// TIA Portal V18 export
DATA_BLOCK "SS1_758A1_16DI_DI_Vars"   // DB11061
{ S7_Optimized_Access := 'FALSE' }
VERSION : 0.1
// stored: AutoNumber false, DBAccessibleFromOPCUA true, IsOnlyStoredInLoadMemory false, IsWriteProtectedInAS false
   VAR
      DI1 : "UDT_DIadv";   // HS Перегрів вн. наос К2 (10.20) термоконтакт
      DI2 : "UDT_DIadv";   // HS Авто режим насосів опалення (10.202+10.203)
      DI3 : "UDT_DIadv";   // HS Несправність насос опалення 1 (10.202)
      DI4 : "UDT_DIadv";   // HS Несправність насос опалення 2 (10.203)
      DI5 : "UDT_DIadv";   // Робота обігріву дизельпроводу
      DI6 : "UDT_DIadv";   // Резерв
      DI7 : "UDT_DIadv";   // Перегрів двигуна тепл. вентиляторів (8.215+8.216)
      DI8 : "UDT_DIadv";   // Робота тепл. вентиляторів (8.215+8.216)
      DI9 { S7_SetPoint := 'True'} : "UDT_DIadv";   // Термостат загр. замерз. (8.73)
      DI10 { S7_SetPoint := 'True'} : "UDT_DIadv";   // Термостат загр. замерз. (8.74)
      DI11 { S7_SetPoint := 'True'} : "UDT_DIadv";   // Несправність цирк. насос (8.217)
      DI12 { S7_SetPoint := 'True'} : "UDT_DIadv";   // Робота цирк. насос (8.217)
      DI13 { S7_SetPoint := 'True'} : "UDT_DIadv";   // Авто режим цирк. насос (8.217)
      DI14 { S7_SetPoint := 'True'} : "UDT_DIadv";   // Забруднення пр. фільтру (8.71)
      DI15 { S7_SetPoint := 'True'} : "UDT_DIadv";   // Забруднення пр. фільтру (8.72)
      DI16 { S7_SetPoint := 'True'} : "UDT_DIadv";   // HS Робота насосу опалення 1 (10.202)
   END_VAR
BEGIN
   DI1.cFuncSystemID := 100;
   DI1.cFuncVar := 1;
   DI2.cFuncSystemID := 100;
   DI2.cFuncVar := 3;
   DI5.cFuncSystemID := 100;
   DI5.cFuncVar := 5;
   DI6.cFuncSystemID := 100;
   DI6.cFuncVar := 6;
END_DATA_BLOCK
